TYPE ST_RecipeBuilder_Config :
    STRUCT
	PanelFrontLength : REAL;
	PanelFrontWidth : REAL;
	PanelHeight : REAL;
	RailHeightCorrection :REAL;
	CuttingOverpass      : REAL;
    GroovingOverpass     : REAL;
    END_STRUCT
END_TYPE

(* stored: Version 1.1.0.1, ProductVersion 3.1.4024.15
   DUT ST_RecipeBuilder_Config: Id {dbdbd64a-f55f-4772-a86a-1207ae4f3c57} *)
